// TwinCAT 3 PLC project TcOscatBasicTests
// Title: TcOscatBasicTests
// Company: Mihai Gînța
// Author: TcOscatBasic developers
// Description: Unit tests for TcOscatBasic, it uses TcUnit and TcOscatBasic as referenced library.
// ProgramVersion: 3.1.4026.22
// libraries:
//   Tc2_Standard, * (Beckhoff Automation GmbH)
//   Tc2_System, * (Beckhoff Automation GmbH)
//   [TcOscatBasic], * (Mihai Gînța)
//   TcUnit, * (www.tcunit.org)
// project tree:
//   / PlcTask.TcTTO
//   TESTs/ FB_B_Trig_Test.TcPOU, FB_String_Test.TcPOU, FB_Version_Test.TcPOU, PRG_TEST.TcPOU
// real-time tasks:
//   TASK PlcTask: cycle T#10ms, priority 21, ADS port 351

CONFIGURATION TcOscatBasicTests
    RESOURCE PLC ON TwinCAT3
        TASK PlcTask(INTERVAL := T#10ms, PRIORITY := 21);
        PROGRAM PRG_TEST WITH PlcTask : PRG_TEST;
    END_RESOURCE
END_CONFIGURATION

// ---- TESTs/PRG_TEST.TcPOU
PROGRAM PRG_TEST
VAR
	String_Test : FB_String_Test;
	B_Trig_Test: FB_B_Trig_Test;
	Version_Test: FB_Version_Test;
END_VAR

TcUnit.RUN();

END_PROGRAM

// ---- TESTs/FB_String_Test.TcPOU
FUNCTION_BLOCK FB_String_Test EXTENDS TcUnit.FB_TestSuite

WhenSubtringExistsExpectPosition();
WhenMonthToStringReturnsCorrectMonthName();
WhenCapitalizeReturnsExpectedResult();
WhenLowercaseReturnsExpectedResult();
WhenUppercaseReturnsExpectedResult();
WhenTrimReturnsExpectedResult();
WhenMirrorReturnsExpectedResult();
WhenCountCharReturnsExpectedResult();
WhenCountSubstringReturnsExpectedResult();
WhenReplaceAllReturnsExpectedResult();
WhenDelCharsReturnsExpectedResult();

METHOD PRIVATE WhenCapitalizeReturnsExpectedResult
VAR
    ActualStr : STRING(20);
    ExpectedStr : STRING(20) := 'Hello World';
    TestStr : STRING(20) := 'hello world';
END_VAR
TEST(__POUNAME());

// @TEST-RUN
ActualStr := CAPITALIZE(TestStr);

// @TEST-ASSERT
AssertEquals_STRING(ExpectedStr, ActualStr, 'CAPITALIZE did not return expected result');

TEST_FINISHED();
END_METHOD

METHOD PRIVATE WhenCountCharReturnsExpectedResult
VAR
    ActualCount : INT;
    ExpectedCount : INT := 3;
    TestStr : STRING(20) := 'banana';
    TestChar : BYTE := 97; // 'a'
END_VAR
TEST(__POUNAME());

// @TEST-RUN
ActualCount := COUNT_CHAR(TestStr, TestChar);

// @TEST-ASSERT
AssertEquals_INT(ExpectedCount, ActualCount, 'COUNT_CHAR did not return expected result');

TEST_FINISHED();
END_METHOD

METHOD PRIVATE WhenCountSubstringReturnsExpectedResult
VAR
    ActualCount : INT;
    ExpectedCount : INT := 2;
    TestStr : STRING(30) := 'the cat sat on the cat';
    SubStr : STRING(10) := 'cat';
END_VAR
TEST(__POUNAME());

// @TEST-RUN
ActualCount := COUNT_SUBSTRING(SubStr, TestStr);

// @TEST-RUN
AssertEquals_INT(ExpectedCount, ActualCount, 'COUNT_SUBSTRING did not return expected result');

TEST_FINISHED();
END_METHOD

METHOD PRIVATE WhenDelCharsReturnsExpectedResult
VAR
    ActualStr : STRING(30);
    ExpectedStr : STRING(30) := 'hll wrld';
    TestStr : STRING(30) := 'hello world';
    CharsToDel : STRING(10) := 'eo';
END_VAR
TEST(__POUNAME());

// @TEST-RUN
ActualStr := DEL_CHARS(TestStr, CharsToDel);

// @TEST-ASSERT
AssertEquals_STRING(ExpectedStr, ActualStr, 'DEL_CHARS did not return expected result');

TEST_FINISHED();
END_METHOD

METHOD PRIVATE WhenLowercaseReturnsExpectedResult
VAR
    ActualStr : STRING(20);
    ExpectedStr : STRING(20) := 'hello world';
    TestStr : STRING(20) := 'HELLO WORLD';
END_VAR
TEST(__POUNAME());

// @TEST-RUN
ActualStr := LOWERCASE(TestStr);

// @TEST-ASSERT
AssertEquals_STRING(ExpectedStr, ActualStr, 'LOWERCASE did not return expected result');

TEST_FINISHED();
END_METHOD

METHOD PRIVATE WhenMirrorReturnsExpectedResult
VAR
    ActualStr : STRING(20);
    ExpectedStr : STRING(20) := 'dlrow olleh';
    TestStr : STRING(20) := 'hello world';
END_VAR
TEST(__POUNAME());

// @TEST-RUN
ActualStr := MIRROR(TestStr);

// @TEST-ASSERT
AssertEquals_STRING(ExpectedStr, ActualStr, 'MIRROR did not return expected result');

TEST_FINISHED();
END_METHOD

METHOD PRIVATE WhenMonthToStringReturnsCorrectMonthName
VAR
    ActualMonth : STRING(10);
    ExpectedMonth : STRING(10) := 'January';
    MTH : INT := 1;
    LANG : INT := 1; // Adjust as needed for your language table
    LX : INT := 0;
END_VAR
TEST(__POUNAME());

// @TEST-RUN
ActualMonth := MONTH_TO_STRING(MTH:=MTH, LANG:=LANG, LX:=LX);

// @TEST-ASSERT
AssertEquals_STRING(ExpectedMonth, ActualMonth, 'MONTH_TO_STRING did not return expected month name');

TEST_FINISHED();
END_METHOD

METHOD PRIVATE WhenReplaceAllReturnsExpectedResult
VAR
    ActualStr : STRING(30);
    ExpectedStr : STRING(30) := 'foo bar foo bar';
    TestStr : STRING(30) := 'foo baz foo baz';
    Src : STRING(10) := 'baz';
    Rep : STRING(10) := 'bar';
END_VAR
TEST(__POUNAME());

// @TEST-RUN
ActualStr := REPLACE_ALL(TestStr, Src, Rep);

// @TEST-ASSERT
AssertEquals_STRING(ExpectedStr, ActualStr, 'REPLACE_ALL did not return expected result');

TEST_FINISHED();
END_METHOD

METHOD PRIVATE WhenSubtringExistsExpectPosition
VAR
	ActualPosition : INT;
	ExpectedPosition : INT := 11;
END_VAR
TEST(__POUNAME());

// @TEST-RUN
ActualPosition := FINDP(str:='Premature optimization is the root of all evil', src:='optimization', pos:=1);

// @TEST-ASSERT
AssertTrue(ActualPosition=ExpectedPosition, 'Substring not found in target string');

TEST_FINISHED();
END_METHOD

METHOD PRIVATE WhenTrimReturnsExpectedResult
VAR
    ActualStr : STRING(20);
    ExpectedStr : STRING(20) := 'helloworld';
    TestStr : STRING(20) := 'hello world';
END_VAR
TEST(__POUNAME());

// @TEST-RUN
ActualStr := TRIM(TestStr);

// @TEST-ASSERT
AssertEquals_STRING(ExpectedStr, ActualStr, 'TRIM did not return expected result');

TEST_FINISHED();
END_METHOD

METHOD PRIVATE WhenUppercaseReturnsExpectedResult
VAR
    ActualStr : STRING(20);
    ExpectedStr : STRING(20) := 'HELLO WORLD';
    TestStr : STRING(20) := 'hello world';
END_VAR
TEST(__POUNAME());

// @TEST-RUN
ActualStr := UPPERCASE(TestStr);

// @TEST-ASSERT
AssertEquals_STRING(ExpectedStr, ActualStr, 'UPPERCASE did not return expected result');

TEST_FINISHED();
END_METHOD

END_FUNCTION_BLOCK

// ---- TESTs/FB_B_Trig_Test.TcPOU
FUNCTION_BLOCK FB_B_Trig_Test EXTENDS TcUnit.FB_TestSuite
VAR
	Trig: B_TRIG;
END_VAR

WhenFallingEdgeExpectCount();
WhenRisingEdgeExpectCount();

METHOD WhenFallingEdgeExpectCount : REFERENCE TO FB_Test
VAR_INPUT
END_VAR
TEST(__POUNAME());

// @TEST-RUN
Trig(CLK:=TRUE);
Trig(CLK:=FALSE);

// @TEST-ASSERT
AssertTrue(Trig.Q, 'B_Trig did not count falling edge');

TEST_FINISHED();
END_METHOD

METHOD WhenRisingEdgeExpectCount
VAR_INPUT
END_VAR
TEST(__POUNAME());

// @TEST-RUN
Trig(CLK:=FALSE);
Trig(CLK:=TRUE);

// @TEST-ASSERT
AssertTrue(Trig.Q, 'B_Trig did not count rising edge');

TEST_FINISHED();
END_METHOD

END_FUNCTION_BLOCK

// ---- TESTs/FB_Version_Test.TcPOU
FUNCTION_BLOCK FB_Version_Test EXTENDS TcUnit.FB_TestSuite

WhenOscatVersionSameAsMajorMinor();

METHOD WhenOscatVersionSameAsMajorMinor : REFERENCE TO FB_Test
VAR
	OscatVersion: DWORD;
	OscatVersionGLobal:DWORD;
END_VAR
TEST(__POUNAME());

// @TEST-RUN
OscatVersion := OSCAT_VERSION(in:=FALSE);
OscatVersionGLobal := TcOscatBasic.Global_Version.stLibVersion_TcOscatBasic.iMajor*100 + TcOscatBasic.Global_Version.stLibVersion_TcOscatBasic.iMinor;

// @TEST-ASSERT
AssertEquals_DWORD(OscatVersion, OscatVersionGLobal, 'Versions do not match');

TEST_FINISHED();
END_METHOD

END_FUNCTION_BLOCK
